PROGRAM MAIN_Control

VAR		
	bValveTest  : BOOL := FALSE;
	timerOnInit : TON;
    bLoadSysParametersExecute : BOOL;
    bLoadSysParametersReset   : BOOL;
END_VAR

timerOnInit(IN := TRUE, PT := T#10S);

//Main Controll
DB_Query();
PRG_MasterControl();
PRG_UpdateVariablesMoving();
PRG_SafetyHandle();
PRG_AxisAssignment();

//MainEvents
POU_EventTest();
POU_FaultHandler();
PRG_MasterSystemTime();

//MainHMI
PRG_HMIControl();
PRG_TowerAlarmLamps();
PRG_LevelHandler();
PRG_ValvePositionRecovery();

//MainServices
PRG_ReportsManager();
PRG_ShutdownPLC();
PRG_RecipeManager();
PRG_SystemInfo();
PRG_UserManagementHistory();

IF timerOnInit.Q
AND NOT DB_Load_SysParameters.bBusy
AND NOT DB_Load_SysParameters.bDone
AND NOT DB_Load_SysParameters.bError THEN
    bLoadSysParametersExecute := TRUE;
END_IF

DB_Load_SysParameters(
    bExecute := bLoadSysParametersExecute,
    bReset   := bLoadSysParametersReset
);

IF DB_Load_SysParameters.bDone OR DB_Load_SysParameters.bError THEN
    bLoadSysParametersExecute := FALSE;
END_IF

// Valve testing
IF bValveTest THEN
	PRG_ValveTest();
END_IF

END_PROGRAM

(* stored: Version 1.1.0.1, ProductVersion 3.1.4024.15
   POU MAIN_Control: Id {cebf6aa5-5e58-48d5-8759-1298446923a5}, SpecialFunc None *)
